        $ 4818 "Until (tool_contact_detection)"
        break
      end
      sync()
    end
    $ 4819 "Direction: Base Z+"
    global move_thread_flag_4819=0
    thread move_thread_4819():
      enter_critical
      move_thread_flag_4819 = 1
      local towardsPos=calculate_point_to_move_towards(p[0.0,0.0,0.0,0.0,0.0,0.0], [0.0,0.0,1.0], 0.08)
      movel(towardsPos, a=0.15, v=0.1)
      move_thread_flag_4819 = 2
      exit_critical
    end
    move_thread_flag_4819 = 0
    move_thread_han_4819 = run move_thread_4819()
    while (True):
      sleep(1.0E-10)
      if (move_thread_flag_4819 > 1):
        join move_thread_han_4819
        $ 4820 "Until (distance)"
        break
      end
      sync()
    end
    $ 4821 "Linea29_B" "breakAfter"
    movel(Linea29_B_p, a=0.5, v=0.1)
    $ 4823 "bajada_comprobacion"
    $ 4824 "Direction: Base Z-"
    global move_thread_flag_4824=0
    thread move_thread_4824():
      enter_critical
      move_thread_flag_4824 = 1
      local towardsPos=calculate_point_to_move_towards(p[0.0,0.0,0.0,0.0,0.0,0.0], [0.0,0.0,-1.0], 0.071)
      movel(towardsPos, a=0.15, v=0.1)
      move_thread_flag_4824 = 2
      exit_critical
    end
    move_thread_flag_4824 = 0
    move_thread_han_4824 = run move_thread_4824()
    while (True):
      sleep(1.0E-10)
      if (move_thread_flag_4824 > 1):
        join move_thread_han_4824
        $ 4825 "Until (distance)"
        break
      end
      sync()
    end
    $ 4826 "Direction: Base Z-"
    global move_thread_flag_4826=0
    thread move_thread_4826():
      enter_critical
      move_thread_flag_4826 = 1
      local towardsPos=calculate_point_to_move_towards(p[0.0,0.0,0.0,0.0,0.0,0.0], [0.0,0.0,-1.0], 1000.0)
      movel(towardsPos, a=0.007, v=0.007)
      move_thread_flag_4826 = 2
      exit_critical
    end
    move_thread_flag_4826 = 0
    move_thread_han_4826 = run move_thread_4826()
    while (True):
      local targetTcpDirection=get_target_tcp_speed()
      local stepsToRetract=tool_contact(direction=targetTcpDirection)
      if (stepsToRetract > 0):
        kill move_thread_han_4826
        stopl(0.02)
        local backTrackMovement=get_actual_joint_positions_history(stepsToRetract)
        local contactPose=get_forward_kin(backTrackMovement)
        local posDir=[targetTcpDirection[0],targetTcpDirection[1],targetTcpDirection[2]]
        local retractTo=contactPose
        if (norm(posDir) > 1e-6):
          local normalizedPosDir=normalize(posDir)
          local additionalRetraction=p[normalizedPosDir[0] * 0.0, normalizedPosDir[1] * 0.0, normalizedPosDir[2] * 0.0, 0, 0, 0]
          retractTo = pose_sub(contactPose, additionalRetraction)
        end
        movel(retractTo, a=0.02, v=0.1)
        $ 4827 "Until (tool_contact_detection)"
        break
      end
      sync()
    end
    $ 4828 "Direction: Base Z+"
    global move_thread_flag_4828=0
    thread move_thread_4828():
      enter_critical
      move_thread_flag_4828 = 1
      local towardsPos=calculate_point_to_move_towards(p[0.0,0.0,0.0,0.0,0.0,0.0], [0.0,0.0,1.0], 0.08)
      movel(towardsPos, a=0.15, v=0.1)
      move_thread_flag_4828 = 2
      exit_critical
    end
    move_thread_flag_4828 = 0
    move_thread_han_4828 = run move_thread_4828()
    while (True):
      sleep(1.0E-10)
      if (move_thread_flag_4828 > 1):
        join move_thread_han_4828
        $ 4829 "Until (distance)"
        break
      end
      sync()
    end
    $ 4830 "AB"
    $ 4831 "'desbaste_inicial'"
    # 'desbaste_inicial'
    $ 4832 "bajada_broca≔p[0,0,-0.008,0,0,0]"
    global bajada_broca=p[0,0,-0.008,0,0,0]
    $ 4833 "barrenos_menos1≔10"
    global barrenos_menos1=10
    $ 4834 "barreno_actual≔5"
    global barreno_actual=5
    $ 4835 "Loop barreno_actual≤barrenos_menos1"
    while (barreno_actual <= barrenos_menos1):
      $ 4836 "Perforacion"
      $ 4837 "MoveL"
      $ 4840 "internos≔interpolate_pose(Linea29_BA, Linea29_B, barreno_actual/barrenos_menos1)"
      global internos= interpolate_pose (Linea29_BA_p, Linea29_B_p, barreno_actual/barrenos_menos1)
      $ 4844 "internos" "breakAfter"
      movel(internos, a=0.5, v=0.1)
      $ 4845 "'desbaste_inicial'"
      # 'desbaste_inicial'
      $ 4846 "bajada_broca≔p[0,0,-0.024,0,0,0]"
      global bajada_broca=p[0,0,-0.024,0,0,0]
      $ 4847 "bajada≔p[0,0,0.024,0,0,0]"
      global bajada=p[0,0,0.024,0,0,0]
      $ 4848 "Direction: Base Z-"
      global move_thread_flag_4848=0
      thread move_thread_4848():
        enter_critical
        move_thread_flag_4848 = 1
        local towardsPos=calculate_point_to_move_towards(p[0.0,0.0,0.0,0.0,0.0,0.0], [0.0,0.0,-1.0], 0.071)
        movel(towardsPos, a=0.15, v=0.1)
        move_thread_flag_4848 = 2
        exit_critical
      end
      move_thread_flag_4848 = 0
      move_thread_han_4848 = run move_thread_4848()
      while (True):
        sleep(1.0E-10)
        if (move_thread_flag_4848 > 1):
          join move_thread_han_4848
          $ 4849 "Until (distance)"
          break
        end
        sync()
      end
      $ 4850 "Direction: Base Z-"
      global move_thread_flag_4850=0
      thread move_thread_4850():
        enter_critical
        move_thread_flag_4850 = 1
        local towardsPos=calculate_point_to_move_towards(p[0.0,0.0,0.0,0.0,0.0,0.0], [0.0,0.0,-1.0], 1000.0)
        movel(towardsPos, a=0.007, v=0.007)
        move_thread_flag_4850 = 2
        exit_critical
      end
      move_thread_flag_4850 = 0
      move_thread_han_4850 = run move_thread_4850()
      while (True):
        local targetTcpDirection=get_target_tcp_speed()
        local stepsToRetract=tool_contact(direction=targetTcpDirection)
        if (stepsToRetract > 0):
          kill move_thread_han_4850
          stopl(0.02)
          local backTrackMovement=get_actual_joint_positions_history(stepsToRetract)
          local contactPose=get_forward_kin(backTrackMovement)
          local posDir=[targetTcpDirection[0],targetTcpDirection[1],targetTcpDirection[2]]
          local retractTo=contactPose
          if (norm(posDir) > 1e-6):
            local normalizedPosDir=normalize(posDir)
            local additionalRetraction=p[normalizedPosDir[0] * 0.0, normalizedPosDir[1] * 0.0, normalizedPosDir[2] * 0.0, 0, 0, 0]
            retractTo = pose_sub(contactPose, additionalRetraction)
          end
          movel(retractTo, a=0.02, v=0.1)
          $ 4851 "Until (tool_contact_detection)"
          break
        end
        sync()
      end
      $ 4852 "Popup: punto contacto alanzdo"
      popup("punto contacto alanzdo", "Mensaje", False, False, blocking=True)
      $ 4853 "Direction: Base Z+"
      global move_thread_flag_4853=0
      thread move_thread_4853():
        enter_critical
        move_thread_flag_4853 = 1
        local towardsPos=calculate_point_to_move_towards(p[0.0,0.0,0.0,0.0,0.0,0.0], [0.0,0.0,1.0], 0.007)
        movel(towardsPos, a=0.015, v=0.015)
        move_thread_flag_4853 = 2
        exit_critical
      end
      move_thread_flag_4853 = 0
      move_thread_han_4853 = run move_thread_4853()
      while (True):
        sleep(1.0E-10)
        if (move_thread_flag_4853 > 1):
          join move_thread_han_4853
          $ 4854 "Until (distance)"
          break
        end
        sync()
      end
      $ 4855 "Wait: 0.3"
      sleep(0.3)
      $ 4856 "Set CO[1]=Encender"
      set_configurable_digital_out(1, True)
      $ 4857 "Wait: 0.3"
      sleep(0.3)
      $ 4858 "Loop 1 times"
      Loop_30 = 0
      while (Loop_30 < 1):
        $ 4859 "bajar≔pose_add(get_actual_tcp_pose(), bajada_broca)"
        global bajar= pose_add ( get_actual_tcp_pose (), bajada_broca)
        $ 4860 "bajar" "breakAfter"
        movel(bajar, a=0.004, v=0.004)
        $ 4861 "subir≔pose_sub(get_actual_tcp_pose(), bajada_broca)"
        global subir= pose_sub ( get_actual_tcp_pose (), bajada_broca)
        $ 4862 "Direction: Base Z+"
        global move_thread_flag_4862=0
        thread move_thread_4862():
          enter_critical
          move_thread_flag_4862 = 1
          local towardsPos=calculate_point_to_move_towards(p[0.0,0.0,0.0,0.0,0.0,0.0], [0.0,0.0,1.0], 0.002)
          movel(towardsPos, a=0.015, v=0.015)
          move_thread_flag_4862 = 2
          exit_critical
        end
        move_thread_flag_4862 = 0
        move_thread_han_4862 = run move_thread_4862()
        while (True):
          sleep(1.0E-10)
          if (move_thread_flag_4862 > 1):
            join move_thread_han_4862
            $ 4863 "Until (distance)"
            break
          end
          sync()
        end
        $ 4864 "Set CO[1]=Apagar"
        set_configurable_digital_out(1, False)
        $ 4865 "subir" "breakAfter"
        movel(subir, a=0.015, v=0.015)
        $ 4866 "bajada_broca≔pose_sub(bajada_broca, bajada)"
        global bajada_broca= pose_sub (bajada_broca, bajada)
        Loop_30 = Loop_30 + 1
      end
      $ 4867 "Direction: Base Z+"
      global move_thread_flag_4867=0
      thread move_thread_4867():
        enter_critical
        move_thread_flag_4867 = 1
        local towardsPos=calculate_point_to_move_towards(p[0.0,0.0,0.0,0.0,0.0,0.0], [0.0,0.0,1.0], 0.04)
        movel(towardsPos, a=0.15, v=0.1)
        move_thread_flag_4867 = 2
        exit_critical
      end
      move_thread_flag_4867 = 0
      move_thread_han_4867 = run move_thread_4867()
      while (True):
        sleep(1.0E-10)
        if (move_thread_flag_4867 > 1):
          join move_thread_han_4867
          $ 4868 "Until (distance)"
          break
        end
        sync()
      end
      $ 4869 "Set CO[1]=Apagar"
      set_configurable_digital_out(1, False)
      $ 4870 "barreno_actual≔barreno_actual+1"
      global barreno_actual=barreno_actual+1
    end
    $ 4873 "Popup: Linea29 con chica Terminada!"
    popup("Linea29 con chica Terminada!", "Mensaje", False, False, blocking=True)
    $ 5361 "'Subprogramas:'"
    # 'Subprogramas:'
  end
end
